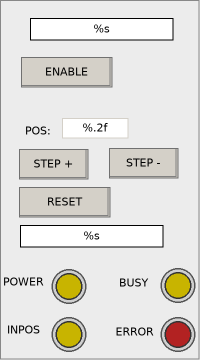
VISUALIZATION vAXIS_CONTROLLER  // 200x360
VAR_IN_OUT
	vAXIS:FB_Axis;
END_VAR
    Rectangle (30,18 143x22), "%s", text variable: vAXIS.sName
    Lamp1 (49,264 40x45), variable: vAxis.power.Enable, style: Lamp-Lamp1-Yellow
    Label (-4,271 55x22), "POWER"
    Lamp1 (49,312 40x45), variable: vAxis.bInPos, style: Lamp-Lamp1-Yellow
    Lamp1 (158,312 40x45), variable: vAxis.bAXIS_ERROR, style: Lamp-Lamp1-Red
    Lamp1 (158,263 40x45), variable: vAxis.bBusy, style: Lamp-Lamp1-Yellow
    Label (-4,319 55x22), "INPOS"
    Label (107,321 55x22), "ERROR"
    Label (106,272 55x22), "BUSY"
    Textfield (62,118 66x20), "%.2f", text variable: vAXIS.Axis.NcToPlc.ActPos
        OnMouseDown: write the text variable via Default
    Label (20,120 36x22), "POS:"
    Button (19,149 69x30), "STEP +"
        OnMouseDown: execute { vAXIS.mMOVE_REL(1000); }
    Button (21,57 91x30), "ENABLE"
        toggle vAxis.bEnable
    Button (19,187 91x30), "RESET"
        OnMouseDown: execute { vAXIS.bReset:=TRUE; }
    Button (109,148 69x30), "STEP -"
        OnMouseDown: execute { vAXIS.mMOVE_REL(-1000); }
    Rectangle (20,225 143x22), "%s", text variable: vAXIS.sAXIS_STATE
END_VISUALIZATION

(* stored: Version 1.1.0.1, ProductVersion 3.1.4024.12
   Visu vAXIS_CONTROLLER: Id {fec02875-7972-421a-a025-805b0db849d4} *)
